// TIA Portal project "Safe" (V16)

(* hardware
DEVICE "S71500/ET200MP station_1"  S7-1500 station
   slot 0: "Rail_0"  Rack  6ES7 590-1***0-0AA0
   slot 1: "PLC_1"  CPU 1511-1 PN  6ES7 511-1AK00-0AB0  V1.8
      slot 3: "CPU display_1"  6ES7591-1AA00-0AA0
      slot 32768: "PROFINET interface_1"  X1
         slot 32769: "Port_1"  X1 P1
         slot 32770: "Port_2"  X1 P2
DEVICE "HMI_1"  KTP1000 Basic color DP
   slot 0: "HMI_1"  KTP1000 Basic color DP  6AV6 647-0AE11-3AX0  12.0.0.0
   slot 1: "HMI_RT_1"  KTP1000 Basic color DP  6AV6 647-0AE11-3AX0  12.0.0.0
   slot 7: "HMI_1.MPI/DP_CP_1"  MPI/DP Interface  12.0.0.0
*)

// ===== PLC "PLC_1"  CPU 1511-1 PN =====

ORGANIZATION_BLOCK "Main"   // OB1, LAD, ProgramCycle
TITLE = "Main Program Sweep (Cycle)"
{ S7_Optimized_Access := 'TRUE' }
VERSION : 0.1
   VAR_INPUT
      Initial_Call : Bool;   // Initial call of this OB
      Remanence : Bool;   // =True, if remanent data are available
   END_VAR
BEGIN
END_ORGANIZATION_BLOCK

(* ===== HMI "HMI_RT_1" =====
system functions are stored by id; their names below are inferred from use

HMI tags "Default tag table"
   "Tag_ScreenNumber" : UInt, internal

Template "Template_1" 640x480
   Button "Exit" at 560,422 size 79x57; TextOff 'Exit'; PictureOff "ExitRuntime_KTP1000_Basic_color_DP"; PictureOn "ExitRuntime_KTP1000_Basic_color_DP"
      on Release: StopRuntime(0)
   Button "Template_Button" at 480,422 size 79x57; TextOff 'Text'
   Button "Template_Button_1" at 400,422 size 79x57; TextOff 'Text'
   Button "Template_Button_2" at 320,422 size 79x57; TextOff 'Text'
   Button "Template_Button_3" at 240,422 size 79x57; TextOff 'Text'
   Button "Template_Button_4" at 160,422 size 79x57; TextOff 'Text'
   Button "Template_Button_5" at 80,422 size 79x57; TextOff 'Text'
   Button "Start screen" at 0,422 size 79x57; TextOff 'Start screen'; PictureOff "NavigateHome_KTP1000_Basic_color_DP"; PictureOn "NavigateHome_KTP1000_Basic_color_DP"
      on Release: ActivateScreen("Root screen", 0)
   SymbolicIOField "Symbolic_IO_Field_Screen" at 105,11 size 428x34; TextOff '0'; TextOn '1'; TextList "TextList_ScreenNames"
      ProcessValue <- "Tag_ScreenNumber"
      on Change: ActivateScreenByNumber("Tag_ScreenNumber", 0)
   DateTimeField "HmiScreenItemData" at 535,29 size 105x29
   DateTimeField "HmiScreenItemData_1" at 535,0 size 105x29
   GraphicView "Logo" at 0,0 size 103x58; Picture "Logo of HMI_1"

screen "Root screen" 640x480, template "Template_1"
   on GenerateScreen: SetTag("Tag_ScreenNumber", 1)
   Button "Button_1" at 435,213 size 36x32; TextOff '1'
      on Press: InvertBit(N)
   Button "Button_2" at 482,213 size 36x32; TextOff '2'
   Button "Button_3" at 529,213 size 36x32; TextOff '3'
   Button "Button_4" at 435,258 size 36x32; TextOff '4'
   Button "Button_5" at 482,258 size 36x32; TextOff '5'
   Button "Button_6" at 529,258 size 36x32; TextOff '6'
   Button "Button_7" at 435,303 size 36x32; TextOff '7'
   Button "Button_8" at 482,303 size 36x32; TextOff '8'
   Button "Button_9" at 529,303 size 36x32; TextOff '9'
   Button "Button_10" at 435,348 size 36x32; TextOff 'C'
   Button "Button_11" at 482,348 size 36x32; TextOff '0'
   Button "Button_12" at 529,348 size 36x32; TextOff 'key'
   IOField "I/O field_1" at 40,212 size 129x28; FormatPattern 1111
   TextField "Text field_1" at 25,95 size 14x18; Text '0'
   TextField "Text field_2" at 54,95 size 10x18; Text '1'
   TextField "Text field_3" at 83,95 size 10x18; Text '2'
   TextField "Text field_4" at 113,95 size 14x18; Text '3'
   TextField "Text field_5" at 142,95 size 10x18; Text '4'
   TextField "Text field_6" at 171,95 size 10x18; Text '5'
   TextField "Text field_7" at 199,95 size 10x18; Text '6'
   TextField "Text field_8" at 227,95 size 10x18; Text '7'
   TextField "Text field_9" at 22,149 size 10x18; Text '8'
   TextField "Text field_10" at 51,149 size 10x18; Text '9'
   TextField "Text field_11" at 80,149 size 18x18; Text '10'
   TextField "Text field_12" at 110,149 size 18x18; Text '11'
   TextField "Text field_13" at 139,149 size 18x18; Text '12'
   TextField "Text field_14" at 168,149 size 18x18; Text '13'
   TextField "Text field_15" at 196,149 size 18x18; Text '14'
   TextField "Text field_16" at 224,149 size 18x18; Text '15'
   IOField "I/O field_2" at 434,159 size 129x28; FormatPattern 999
*)